FUNCTION_BLOCK E_TimeOut (* Simple implementation of the timeout services *)
  (* Standard: 61499-2; Description: TODO for efficience reasons make this a service interface FB *)
  (* Version 1.0, 2012-12-18, AZ, 4DIAC-Consortium *)
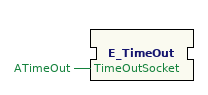
  SOCKETS
    TimeOutSocket : ATimeOut;
  END_SOCKETS
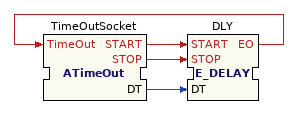
  FBS
    DLY : E_DELAY;
  END_FBS
  EVENT_CONNECTIONS
    TimeOutSocket.START TO DLY.START;
    TimeOutSocket.STOP TO DLY.STOP;
    DLY.EO TO TimeOutSocket.TimeOut;
  END_CONNECTIONS
  DATA_CONNECTIONS
    TimeOutSocket.DT TO DLY.DT;
  END_CONNECTIONS
  SERVICE eTimeOut_interface/eTimeOut_implementation (* Simple implementation of the timeout services *)
    SEQUENCE DelayTime
      eTimeOut_interface.TimeOutSocket.START();
      eTimeOut_interface.TimeOutSocket.START();
      -> eTimeOut_interface.TimeOutSocket.TimeOut();
    END_SEQUENCE
    SEQUENCE DelayStop
      eTimeOut_interface.TimeOutSocket.STOP();
    END_SEQUENCE
  END_SERVICE
END_FUNCTION_BLOCK
